{attribute 'qualified_only'}
{attribute 'strict'}
TYPE DeviceState :
(
	DeviceInINIT,
	DeviceInPREOP,
	DeviceInBOOT,
	DeviceInSAFEOP,
	DeviceInOP
):= DeviceInINIT;
END_TYPE

(* stored: Version 1.1.0.1, ProductVersion 3.1.4024.11
   DUT DeviceState: Id {5365075f-a8e9-4487-bbb9-594e5c3dcb05} *)
